# EPICS substitutions: MX_E12xx_ModbusIOCApp/Db/ioLogik_E1210.substitutions
# ##############################################################################
# ##############################################################################

# asyn record for the underlying asyn octet port
file "$(ASYN)/db/asynRecord.db" { pattern
{P,R, PORT, ADDR,    IMAX,    OMAX}
{"\$(NAME):", "\$(ASYNPORT)_OctetAsyn", "\$(ASYNPORT)",   0,      80,     80}
}

# ##############################################################################
# DIs in "DI mode" (default)
# ##############################################################################

file "bi_bit.template" { pattern
{P,           R,         PORT,           OFFSET,   ZNAM,   ONAM,  ZSV,       OSV,    SCAN}
{"\$(NAME):", "\$(ASYNPORT)_DI_CH00",     "\$(ASYNPORT)_DI",     0x00,        Low,    High,  NO_ALARM,  NO_ALARM,  "I/O Intr"}
{"\$(NAME):", "\$(ASYNPORT)_DI_CH01",     "\$(ASYNPORT)_DI",     0x01,        Low,    High,  NO_ALARM,  NO_ALARM,  "I/O Intr"}
{"\$(NAME):", "\$(ASYNPORT)_DI_CH02",     "\$(ASYNPORT)_DI",     0x02,        Low,    High,  NO_ALARM,  NO_ALARM,  "I/O Intr"}
{"\$(NAME):", "\$(ASYNPORT)_DI_CH03",     "\$(ASYNPORT)_DI",     0x03,        Low,    High,  NO_ALARM,  NO_ALARM,  "I/O Intr"}
{"\$(NAME):", "\$(ASYNPORT)_DI_CH04",     "\$(ASYNPORT)_DI",     0x04,        Low,    High,  NO_ALARM,  NO_ALARM,  "I/O Intr"}
{"\$(NAME):", "\$(ASYNPORT)_DI_CH05",     "\$(ASYNPORT)_DI",     0x05,        Low,    High,  NO_ALARM,  NO_ALARM,  "I/O Intr"}
{"\$(NAME):", "\$(ASYNPORT)_DI_CH06",     "\$(ASYNPORT)_DI",     0x06,        Low,    High,  NO_ALARM,  NO_ALARM,  "I/O Intr"}
{"\$(NAME):", "\$(ASYNPORT)_DI_CH07",     "\$(ASYNPORT)_DI",     0x07,        Low,    High,  NO_ALARM,  NO_ALARM,  "I/O Intr"}
{"\$(NAME):", "\$(ASYNPORT)_DI_CH08",     "\$(ASYNPORT)_DI",     0x08,        Low,    High,  NO_ALARM,  NO_ALARM,  "I/O Intr"}
{"\$(NAME):", "\$(ASYNPORT)_DI_CH09",     "\$(ASYNPORT)_DI",     0x09,        Low,    High,  NO_ALARM,  NO_ALARM,  "I/O Intr"}
{"\$(NAME):", "\$(ASYNPORT)_DI_CH10",     "\$(ASYNPORT)_DI",     0x0A,       Low,    High,  NO_ALARM,  NO_ALARM,  "I/O Intr"}
{"\$(NAME):", "\$(ASYNPORT)_DI_CH11",     "\$(ASYNPORT)_DI",     0x0B,       Low,    High,  NO_ALARM,  NO_ALARM,  "I/O Intr"}
{"\$(NAME):", "\$(ASYNPORT)_DI_CH12",     "\$(ASYNPORT)_DI",     0x0C,       Low,    High,  NO_ALARM,  NO_ALARM,  "I/O Intr"}
{"\$(NAME):", "\$(ASYNPORT)_DI_CH13",     "\$(ASYNPORT)_DI",     0x0D,       Low,    High,  NO_ALARM,  NO_ALARM,  "I/O Intr"}
{"\$(NAME):", "\$(ASYNPORT)_DI_CH14",     "\$(ASYNPORT)_DI",     0x0E,       Low,    High,  NO_ALARM,  NO_ALARM,  "I/O Intr"}
{"\$(NAME):", "\$(ASYNPORT)_DI_CH15",     "\$(ASYNPORT)_DI",     0x0F,       Low,    High,  NO_ALARM,  NO_ALARM,  "I/O Intr"}
}
